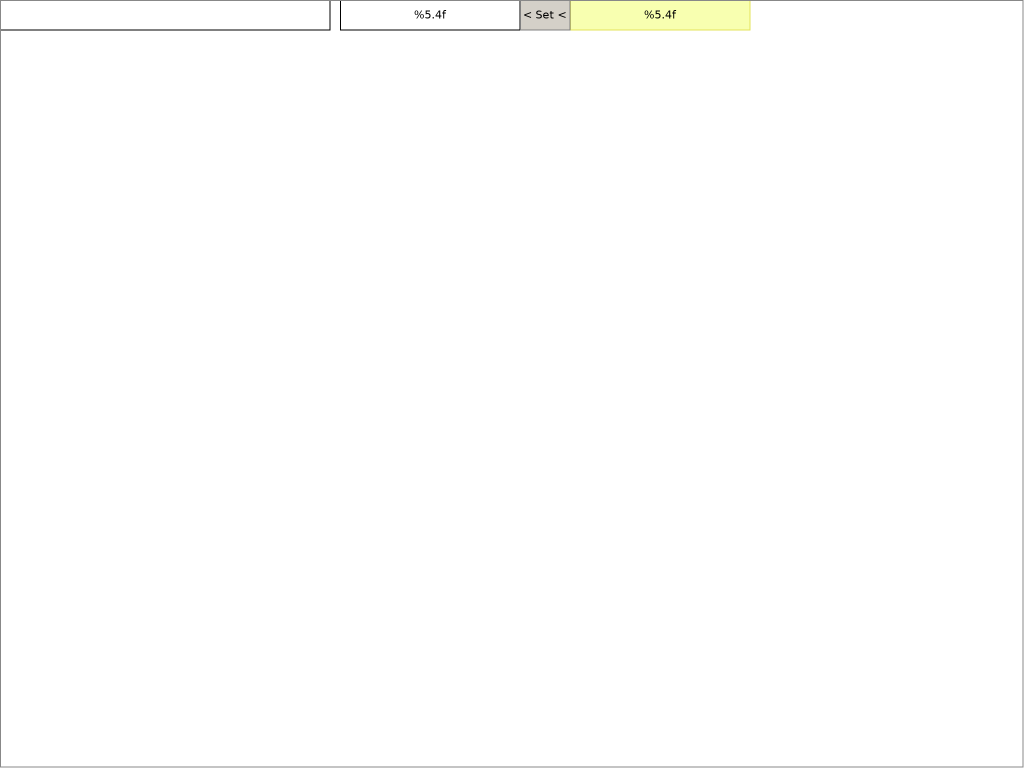
VISUALIZATION Param_LREAL  // 1024x768
VAR_INPUT
	nIdx:		INT;
END_VAR
    Rectangle (340,0 180x30), "%5.4f", text variable: stMParam_Visu.fLrealAktValue[nIdx]
    Rectangle (0,0 330x30), text list: 'TL_Mparams_LREAL', text index: nIdx
    Rectangle (570,0 180x30), "%5.4f", text variable: stMParam_Visu.fLrealNewValue[nIdx]
        OnMouseClick: write the text variable via Default
    Rectangle (520,0 50x30), "< Set <"
        OnMouseClick: execute { stMParam_Visu.bLrealSetValue[nIdx]:=TRUE; }
END_VISUALIZATION

(* stored: Version 1.1.0.1
   Visu Param_LREAL: Id {f839f6a8-a838-4965-8c1e-b04be0835ba4} *)
